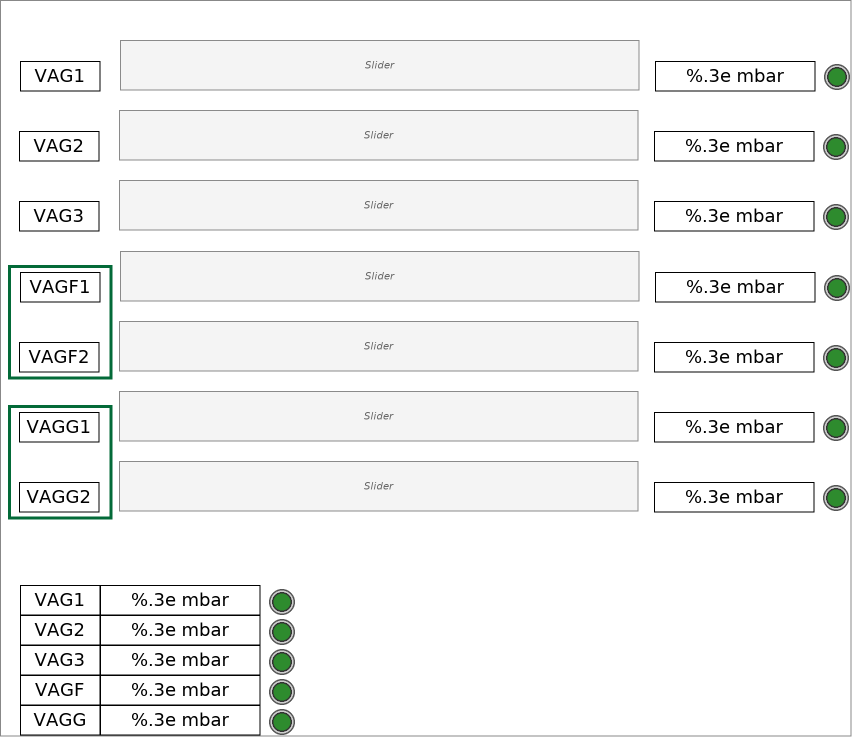
VISUALIZATION GUI_Pressures  // 852x737
    Slider (120,40 519x50), variable: MAIN.q_nVAG1, scale 0..35000
    Rectangle (20,61 80x30), "VAG1"
    Rectangle (655,61 160x30), "%.3e mbar", text variable: MAIN.evac_micado.VAG1.stat.lrPressure
    Lamp1 (822,62 30x30), variable: MAIN.evac_micado.VAG1.stat.bValid, style: Lamp-Lamp1-Green
    Slider (119,110 519x50), variable: MAIN.q_nVAG2, scale 0..35000
    Rectangle (19,131 80x30), "VAG2"
    Rectangle (654,131 160x30), "%.3e mbar", text variable: MAIN.evac_micado.VAG2.stat.lrPressure
    Lamp1 (821,132 30x30), variable: MAIN.evac_micado.VAG2.stat.bValid, style: Lamp-Lamp1-Green
    Slider (119,180 519x50), variable: MAIN.q_nVAG3, scale 0..35000
    Rectangle (19,201 80x30), "VAG3"
    Rectangle (654,201 160x30), "%.3e mbar", text variable: MAIN.evac_micado.VAG3.stat.lrPressure
    Lamp1 (821,202 30x30), variable: MAIN.evac_micado.VAG3.stat.bValid, style: Lamp-Lamp1-Green
    Slider (120,251 519x50), variable: MAIN.q_nVAGF1, scale 0..35000
    Rectangle (20,272 80x30), "VAGF1"
    Rectangle (655,272 160x30), "%.3e mbar", text variable: MAIN.sensor_VAGF1.stat.lrPressure
    Lamp1 (822,273 30x30), variable: MAIN.sensor_VAGF1.stat.bValid, style: Lamp-Lamp1-Green
    Slider (119,321 519x50), variable: MAIN.q_nVAGF2, scale 0..35000
    Rectangle (19,342 80x30), "VAGF2"
    Rectangle (654,342 160x30), "%.3e mbar", text variable: MAIN.sensor_VAGF2.stat.lrPressure
    Lamp1 (821,343 30x30), variable: MAIN.sensor_VAGF2.stat.bValid, style: Lamp-Lamp1-Green
    Slider (119,391 519x50), variable: MAIN.q_nVAGG1, scale 0..35000
    Rectangle (19,412 80x30), "VAGG1"
    Rectangle (654,412 160x30), "%.3e mbar", text variable: MAIN.sensor_VAGG1.stat.lrPressure
    Lamp1 (821,413 30x30), variable: MAIN.sensor_VAGG1.stat.bValid, style: Lamp-Lamp1-Green
    Slider (119,461 519x50), variable: MAIN.q_nVAGG2, scale 0..35000
    Rectangle (19,482 80x30), "VAGG2"
    Rectangle (654,482 160x30), "%.3e mbar", text variable: MAIN.sensor_VAGG2.stat.lrPressure
    Lamp1 (821,483 30x30), variable: MAIN.sensor_VAGG2.stat.bValid, style: Lamp-Lamp1-Green
    Rectangle (20,585 80x30), "VAG1"
    Rectangle (20,615 80x30), "VAG2"
    Rectangle (20,645 80x30), "VAG3"
    Rectangle (100,585 160x30), "%.3e mbar", text variable: MAIN.evac_micado.VAG1.stat.lrPressure
    Lamp1 (267,587 30x30), variable: MAIN.evac_micado.VAG1.stat.bValid, style: Lamp-Lamp1-Green
    Rectangle (100,615 160x30), "%.3e mbar", text variable: MAIN.evac_micado.VAG2.stat.lrPressure
    Lamp1 (267,617 30x30), variable: MAIN.evac_micado.VAG2.stat.bValid, style: Lamp-Lamp1-Green
    Rectangle (100,645 160x30), "%.3e mbar", text variable: MAIN.evac_micado.VAG3.stat.lrPressure
    Lamp1 (267,647 30x30), variable: MAIN.evac_micado.VAG3.stat.bValid, style: Lamp-Lamp1-Green
    Rectangle (20,675 80x30), "VAGF"
    Rectangle (100,675 160x30), "%.3e mbar", text variable: MAIN.evac_micado.VAGF.stat.lrPressure
    Lamp1 (267,677 30x30), variable: MAIN.evac_micado.VAGF.stat.bValid, style: Lamp-Lamp1-Green
    Rectangle (20,705 80x30), "VAGG"
    Rectangle (100,705 160x30), "%.3e mbar", text variable: MAIN.evac_micado.VAGG.stat.lrPressure
    Lamp1 (267,707 30x30), variable: MAIN.evac_micado.VAGG.stat.bValid, style: Lamp-Lamp1-Green
    Rectangle (8,265 104x114)
    Rectangle (8,405 104x114)
END_VISUALIZATION

(* stored: Version 1.1.0.1, ProductVersion 3.1.4024.9
   Visu GUI_Pressures: Id {ab62cca2-decf-4fc3-af9e-4d1c2657b407} *)
